// TIA Portal V20 export
DATA_BLOCK "GDB_ActiveRecipe"   // DB24
TITLE = Active recipes (Modules D+E, dual-pallet, PSC-bound)
{ S7_Optimized_Access := 'TRUE' }
// SCARA Phase 2 Module D + E active-recipe DB (V3.0, 2026-05-23). Two pallet slots (recipe1 = LEFT, recipe2 = RIGHT), each a UDT_Recipe. PSC binds member-for-member to recipe1.* and recipe2.* from separate HMI parameter sets. Pallet selection is operator-driven via the maintained bo_ExecutePallet1 / bo_ExecutePallet2 flags (WanErXin pattern -- no auto-advance); FB_PatternAutoGen mediates the mutex, picks the active recipe, writes its config to GDB_PalletizingCmd, validates both recipes independently, and latches per-pallet bo_PalletNFull alarms on cycle completion attributed to the IN-FLIGHT pallet (snapshotted at cycle start, so mid-cycle operator swaps cannot mis-attribute). Operator swaps pallets by clearing one flag and setting the other -- the just-emptied side's full bit auto-clears so it can be re-used. V3.0 also adds explicit per-pallet bo_AckPalletNFull reset bits and the bo_BothPalletsFull aggregate for HMI / future module integration.
// stored: MemoryReserve 100
   VAR
      recipe1 : "UDT_Recipe";   // Active recipe for PALLET 1 (LEFT). PSC binds and writes here from the HMI's pallet-1 parameter set. FB_PatternAutoGen consumes this each scan iff recipe1.bo_Valid is TRUE AND i16_ActivePalletIdx = 1. StartValues = the verified 16-box 4x(2x2) Module D default.
      recipe2 : "UDT_Recipe";   // Active recipe for PALLET 2 (RIGHT). PSC binds and writes here from the HMI's pallet-2 parameter set. FB_PatternAutoGen consumes this each scan iff recipe2.bo_Valid is TRUE AND i16_ActivePalletIdx = 2. StartValues match recipe1 (pallets share a default product); operator overrides via PSC if pallet 2 should carry a different box product.
      bo_PatternValid1 : Bool;   // FB_PatternAutoGen status for PALLET 1: recipe1 passed validation and its computed grid is mathematically valid. HMI lamp. (Independent of whether pallet 1 is currently active.)
      bo_PatternValid2 : Bool;   // FB_PatternAutoGen status for PALLET 2: recipe2 passed validation.
      bo_PatternError1 : Bool;   // FB_PatternAutoGen status for PALLET 1: recipe1 failed validation. HMI alarm.
      bo_PatternError2 : Bool;   // FB_PatternAutoGen status for PALLET 2: recipe2 failed validation.
      i16_ComputedGridColsX1 : Int;   // FB_PatternAutoGen echo for PALLET 1: auto-fitted columns along X.
      i16_ComputedGridColsX2 : Int;   // FB_PatternAutoGen echo for PALLET 2: auto-fitted columns along X.
      i16_ComputedGridRowsY1 : Int;   // FB_PatternAutoGen echo for PALLET 1: auto-fitted rows along Y.
      i16_ComputedGridRowsY2 : Int;   // FB_PatternAutoGen echo for PALLET 2: auto-fitted rows along Y.
      i16_ComputedBoxCount1 : Int;   // FB_PatternAutoGen echo for PALLET 1: total boxes = Cols x Rows x LayerCount. Must stay within the GDB_PalletizingPath.aCmd[] ceiling (22) or recipe1 is rejected.
      i16_ComputedBoxCount2 : Int;   // FB_PatternAutoGen echo for PALLET 2: total boxes. Same ceiling.
      bo_ExecutePallet1 : Bool := TRUE;   // Operator flag (HMI MAINTAINED button) -- "execute pallet 1" (WanErXin pattern). Setting TRUE while bo_ExecutePallet2=FALSE selects pallet 1 as active; FB_PatternAutoGen then writes recipe1 into GDB_PalletizingCmd. Cleared TRUE by operator releasing the button OR auto-cleared by FB when bo_Pallet1Full (operator must press the other side's button to swap, which auto-clears the just-emptied pallet's full bit so it can be re-used).
      bo_ExecutePallet2 : Bool := FALSE;   // Operator flag -- "execute pallet 2". Mirror of bo_ExecutePallet1 for the right-side pallet. Both flags simultaneously TRUE = mutex stalemate (FB keeps the current active pallet); both FALSE = i16_ActivePalletIdx := 0, no pallet active, GDB_PalletizingCmd left at safe defaults.
      i16_ActivePalletIdx : Int;   // FB_PatternAutoGen status: which pallet is currently active. 1 = pallet 1 (LEFT), 2 = pallet 2 (RIGHT), 0 = neither (no operator flag set OR active recipe invalid). HMI display.
      bo_Pallet1Full : Bool;   // Latched "pallet 1 full" alarm. Set TRUE by FB_PatternAutoGen when GDB_PalletizingCmd.bo_PalletDone is TRUE while i16_ActivePalletIdx = 1 (the cycle just placed the last box of pallet 1). Cleared automatically when the operator switches to pallet 2 (bo_ExecutePallet1 := FALSE AND bo_ExecutePallet2 := TRUE) -- which is interpreted as "I have emptied pallet 1, ready to re-use it later". HMI lamp/alarm.
      bo_Pallet2Full : Bool;   // Latched "pallet 2 full" alarm. Same logic as bo_Pallet1Full, mirrored.
      bo_AckPallet1Full : Bool;   // V3.0 (2026-05-23): Operator acknowledge / explicit reset for bo_Pallet1Full. HMI MAINTAINED button. While TRUE, FB_PatternAutoGen forces bo_Pallet1Full := FALSE every scan -- explicit reset path used when operator has physically emptied pallet 1 and wants to re-use it WITHOUT first having to swap to pallet 2. (The WanErXin swap-clear path remains as a convenience: pressing pallet 2's button while pallet 1's full bit is latched still clears it.) Operator releases the Ack button before re-starting the cycle so the next bo_PalletDone can re-latch bo_Pallet1Full normally.
      bo_AckPallet2Full : Bool;   // V3.0: Operator acknowledge / explicit reset for bo_Pallet2Full. Mirror of bo_AckPallet1Full.
      bo_BothPalletsFull : Bool;   // V3.0: FB-computed aggregate = bo_Pallet1Full AND bo_Pallet2Full. Single status bit for HMI / future Module F-G integration to gate "both pallets need unloading, robot should idle". Read-only from HMI side -- FB_PatternAutoGen is sole writer.
   END_VAR
BEGIN
   recipe1.sName := 'Pallet 1 Default 4x2x2';
   recipe1.bo_Valid := TRUE;
   recipe1.product.lr_Length := 400.0;
   recipe1.product.lr_Width := 600.0;
   recipe1.product.lr_Height := 200.0;
   recipe1.product.lr_Gap := 0.0;
   recipe1.pallet.lr_BaseLength := 800.0;
   recipe1.pallet.lr_BaseWidth := 1200.0;
   recipe1.pallet.i16_LayerCount := 4;
   recipe1.dynamics.lr_Velocity := 2000.0;
   recipe1.dynamics.lr_Acceleration := 10000.0;
   recipe1.dynamics.lr_Deceleration := 10000.0;
   recipe1.dynamics.lr_Jerk := 100000.0;
   recipe2.sName := 'Pallet 2 Default 4x2x2';
   recipe2.bo_Valid := TRUE;
   recipe2.product.lr_Length := 400.0;
   recipe2.product.lr_Width := 600.0;
   recipe2.product.lr_Height := 200.0;
   recipe2.product.lr_Gap := 0.0;
   recipe2.pallet.lr_BaseLength := 800.0;
   recipe2.pallet.lr_BaseWidth := 1200.0;
   recipe2.pallet.i16_LayerCount := 4;
   recipe2.dynamics.lr_Velocity := 2000.0;
   recipe2.dynamics.lr_Acceleration := 10000.0;
   recipe2.dynamics.lr_Deceleration := 10000.0;
   recipe2.dynamics.lr_Jerk := 100000.0;
END_DATA_BLOCK
